TYPE TcaSegmentDoorService :
STRUCT

END_STRUCT
END_TYPE

(* stored: Version 1.1.0.1
   DUT TcaSegmentDoorService: Id {b81e6734-f89a-4e90-9130-0eec935e5c68} *)
